FUNCTION_BLOCK ABSTRACT FB_DriveBase IMPLEMENTS I_DriveBase
VAR
	lrMax : LREAL;
	lrMin : LREAL;
END_VAR

METHOD ABSTRACT Disable : BOOL
END_METHOD

METHOD ABSTRACT Enable : BOOL
END_METHOD

METHOD ABSTRACT MoveToPosition : BOOL
END_METHOD

METHOD ABSTRACT Reset : BOOL
END_METHOD

METHOD SetLimits : BOOL
VAR_INPUT
	lrMax : LREAL;
	lrMin : LREAL;
END_VAR
THIS^.lrMax := lrMax;
THIS^.lrMin := lrMin;
END_METHOD

END_FUNCTION_BLOCK

(* stored: Version 1.1.0.1, ProductVersion 3.1.4024.6
   POU FB_DriveBase: Id {4d2f1c8d-895c-418c-8f96-0fabbe561d56}, SpecialFunc None
   Method Disable: Id {668eefdb-e959-4e3f-9ab3-0785be03ca9c}
   Method Enable: Id {89143ded-6182-4dc9-a443-4edaf6b9890b}
   Method MoveToPosition: Id {097da37f-8ebd-46e9-975d-dfcdce4bea85}
   Method Reset: Id {c73a9d9b-f580-4808-83bd-dd61e45bd4e2}
   Method SetLimits: Id {ec98029c-30bb-4562-8add-ff055a55188f} *)
